{attribute 'enable_dynamic_creation'}
FUNCTION_BLOCK ElectricAdapterMotor EXTENDS Motor
VAR
	pElectricEngine : POINTER TO ElectricMotor;
END_VAR

METHOD FB_exit : BOOL
VAR_INPUT
	bInCopyCode : BOOL; // if TRUE, the exit method is called for exiting an instance that is copied afterwards (online change).
END_VAR
__DELETE (pElectricEngine);
END_METHOD


METHOD FB_init : BOOL
VAR_INPUT
	bInitRetains : BOOL; // if TRUE, the retain variables are initialized (warm start / cold start)
	bInCopyCode : BOOL;  // if TRUE, the instance afterwards gets moved into the copy code (online change)
END_VAR
pElectricEngine := __NEW(ElectricMotor);
END_METHOD

METHOD PUBLIC LoadFuel
pElectricEngine^.Plug();
END_METHOD

METHOD PUBLIC SpeedUp
pElectricEngine^.Travel();
END_METHOD

METHOD PUBLIC StartUp
pElectricEngine^.Connect();
pElectricEngine^.Activate();
END_METHOD

METHOD PUBLIC Stop
pElectricEngine^.Deactivate();
pElectricEngine^.Stop();
END_METHOD

END_FUNCTION_BLOCK

(* stored: Version 1.1.0.1, ProductVersion 3.1.4024.12
   POU ElectricAdapterMotor: Id {b69eb29b-3558-46ff-b1f1-f25e269725c2}, SpecialFunc None
   Method FB_exit: Id {845c3ac7-e64b-4656-bd7f-909a551f9694}
   Method FB_init: Id {6c724098-dd2e-42cc-8617-7b0fce3758be}
   Method LoadFuel: Id {730b5226-e1b4-4962-a3d3-9d07151c17f2}
   Method SpeedUp: Id {9641755b-0306-4223-a9ab-e3a4b3dbcda5}
   Method StartUp: Id {b54191ab-3f4d-472b-a836-aba66da3a43f}
   Method Stop: Id {09b6fda3-fff6-431f-8dcd-03f11369fa2d} *)
